// TwinCAT 3 PLC project Motion_Lib
// Title: Motion Library
// Company: Beckhoff UK
// Author: Chris Knight
// ProjectVersion: 4.1.1
// ProgramVersion: 3.1.4026.25
// libraries:
//   Base Library, * (Beckhoff UK)
//   Tc2_MC2, * (Beckhoff Automation GmbH)
//   Tc2_MC2_Drive, * (Beckhoff Automation GmbH)
//   Tc2_Standard, * (Beckhoff Automation GmbH)
//   Tc2_System, * (Beckhoff Automation GmbH)
//   Tc3_Module, * (Beckhoff Automation GmbH)
// project tree:
//   Axis Class/ Axis_Base.TcPOU
//   Interfaces/ I_Axis.TcIO, I_AxisBase.TcIO, I_Status.TcIO, I_Jog.TcIO, I_Position.TcIO, I_Velocity.TcIO
//   Internal/ I_MoveAbs.TcIO, I_MoveMod.TcIO (not stored), I_MoveRel.TcIO, I_MoveVelo.TcIO, MoveAbs.TcPOU, MoveMod.TcPOU, MoveRel.TcPOU, MoveVelo.TcPOU
//   Operations/ GearAxes.TcPOU
//   Project Information/ F_GetCompany.TcPOU, F_GetTitle.TcPOU, F_GetVersion.TcPOU
//   Tasks/ MoveModTask.TcPOU, MoveRelTask.TcPOU, JogTask.TcPOU, CoEResetTask.TcPOU, EnableDisableTask.TcPOU, HaltTask.TcPOU, MoveVeloTask.TcPOU, MoveAbsTask.TcPOU, SoEResetTask.TcPOU
//   Version/ Global_Version.TcGVL

// ---- Version/Global_Version.TcGVL
{attribute 'TcGenerated'}
{attribute 'no-analysis'}
{attribute 'linkalways'}
// This function has been automatically generated from the project information.
VAR_GLOBAL CONSTANT
	{attribute 'const_non_replaced'}
	stLibVersion_Motion_Library : ST_LibVersion := (iMajor := 4, iMinor := 1, iBuild := 1, iRevision := 0, nFlags := 0, sVersion := '4.1.1');
END_VAR

// ---- Interfaces/I_Axis.TcIO
INTERFACE I_Axis EXTENDS I_Cyclic

PROPERTY PUBLIC Acceleration : mc_lreal
GET
END_GET
SET
END_SET
END_PROPERTY

PROPERTY AxisRef : reference to Axis_Ref
GET
END_GET
END_PROPERTY

PROPERTY BufferMode : MC_BufferMode
GET
END_GET
SET
END_SET
END_PROPERTY

PROPERTY PUBLIC Deceleration : mc_lreal
GET
END_GET
SET
END_SET
END_PROPERTY

METHOD PUBLIC DisableAxis : HRESULT
VAR_INPUT
END_VAR
END_METHOD

METHOD PUBLIC EnableAxis : HRESULT
VAR_INPUT
	InhibitPositive : BOOL;
	InhibitNegative : BOOL;
END_VAR
END_METHOD

PROPERTY ErrorID : DWORD
GET
END_GET
END_PROPERTY

METHOD PUBLIC HaltAxis : HRESULT
VAR
END_VAR
END_METHOD

PROPERTY PUBLIC Jerk : mc_lreal
GET
END_GET
SET
END_SET
END_PROPERTY

PROPERTY Operating : BOOL
GET
END_GET
END_PROPERTY

METHOD PUBLIC Reset : HRESULT
VAR
END_VAR
END_METHOD

END_INTERFACE

// ---- Interfaces/I_AxisBase.TcIO
INTERFACE I_AxisBase EXTENDS I_Axis, I_Status

END_INTERFACE

// ---- Interfaces/I_Status.TcIO
INTERFACE I_Status EXTENDS __SYSTEM.IQueryInterface

PROPERTY CurrentPosition : LREAL
GET
END_GET
END_PROPERTY

PROPERTY CurrentVelocity : LREAL
GET
END_GET
END_PROPERTY

PROPERTY ErrorID : DWORD
GET
END_GET
END_PROPERTY

PROPERTY HasError : BOOL
GET
END_GET
END_PROPERTY

PROPERTY InTargetPosition : BOOL
GET
END_GET
END_PROPERTY

PROPERTY InVelocity : BOOL
GET
END_GET
END_PROPERTY

PROPERTY IsCoupled : bool
GET
END_GET
END_PROPERTY

PROPERTY IsEnabled : bool
GET
END_GET
END_PROPERTY

PROPERTY IsStationary : bool
GET
END_GET
END_PROPERTY

END_INTERFACE

// ---- Interfaces/I_Jog.TcIO
INTERFACE I_Jog EXTENDS I_Axis

METHOD Inch : HRESULT
VAR_INPUT
	Distance : MC_LREAL;
	Direction : BOOL;
END_VAR
END_METHOD

METHOD JogFast : HRESULT
VAR_INPUT
	Direction : BOOL;
END_VAR
END_METHOD

METHOD JogSlow : HRESULT
VAR_INPUT
	Direction : BOOL;
END_VAR
END_METHOD

END_INTERFACE

// ---- Interfaces/I_Position.TcIO
INTERFACE I_Position EXTENDS __SYSTEM.IQueryInterface

PROPERTY CurrentPosition : LREAL
GET
END_GET
END_PROPERTY

PROPERTY IsStationary : bool
GET
END_GET
END_PROPERTY

METHOD MoveByDistance : HRESULT
VAR_INPUT
	Distance : MC_LREAL;
	Velocity : MC_LREAL;
END_VAR
END_METHOD

METHOD MoveToModuloPosition : HRESULT
VAR_INPUT
	Position : MC_LREAL;
	Velocity : MC_LREAL;
END_VAR
END_METHOD

METHOD MoveToPosition : HRESULT
VAR_INPUT
	Position : MC_LREAL;
	Velocity : MC_LREAL;
END_VAR
END_METHOD

END_INTERFACE

// ---- Interfaces/I_Velocity.TcIO
INTERFACE I_Velocity

PROPERTY InVelocity : BOOL
GET
END_GET
END_PROPERTY

METHOD MoveAtVelocity : HRESULT
VAR_INPUT
	Direction : MC_Direction;
	Velocity : MC_LREAL;
END_VAR
END_METHOD

END_INTERFACE

// ---- Internal/I_MoveAbs.TcIO
INTERFACE I_MoveAbs

PROPERTY Acceleration : MC_LREAL
GET
END_GET
SET
END_SET
END_PROPERTY

PROPERTY BufferMode : MC_Buffermode
GET
END_GET
SET
END_SET
END_PROPERTY

PROPERTY Busy : BOOL
GET
END_GET
END_PROPERTY

PROPERTY Deceleration : MC_LREAL
GET
END_GET
SET
END_SET
END_PROPERTY

PROPERTY Done : BOOL
GET
END_GET
END_PROPERTY

PROPERTY Error : BOOL
GET
END_GET
END_PROPERTY

PROPERTY Execute : BOOL
GET
END_GET
SET
END_SET
END_PROPERTY

PROPERTY Jerk : MC_LREAL
GET
END_GET
SET
END_SET
END_PROPERTY

PROPERTY Position : MC_LREAL
GET
END_GET
SET
END_SET
END_PROPERTY

PROPERTY Velocity : MC_LREAL
GET
END_GET
SET
END_SET
END_PROPERTY

END_INTERFACE

// ---- Internal/I_MoveRel.TcIO
INTERFACE I_MoveRel

PROPERTY Acceleration : MC_LREAL
GET
END_GET
SET
END_SET
END_PROPERTY

PROPERTY BufferMode : MC_Buffermode
GET
END_GET
SET
END_SET
END_PROPERTY

PROPERTY Busy : BOOL
GET
END_GET
END_PROPERTY

PROPERTY Deceleration : MC_LREAL
GET
END_GET
SET
END_SET
END_PROPERTY

PROPERTY Distance : MC_LREAL
GET
END_GET
SET
END_SET
END_PROPERTY

PROPERTY Done : BOOL
GET
END_GET
END_PROPERTY

PROPERTY Error : BOOL
GET
END_GET
END_PROPERTY

PROPERTY Execute : BOOL
GET
END_GET
SET
END_SET
END_PROPERTY

PROPERTY Jerk : MC_LREAL
GET
END_GET
SET
END_SET
END_PROPERTY

PROPERTY Velocity : MC_LREAL
GET
END_GET
SET
END_SET
END_PROPERTY

END_INTERFACE

// ---- Internal/I_MoveVelo.TcIO
INTERFACE I_MoveVelo

PROPERTY Acceleration : MC_LREAL
GET
END_GET
SET
END_SET
END_PROPERTY

PROPERTY BufferMode : MC_Buffermode
GET
END_GET
SET
END_SET
END_PROPERTY

PROPERTY Busy : BOOL
GET
END_GET
END_PROPERTY

PROPERTY Deceleration : MC_LREAL
GET
END_GET
SET
END_SET
END_PROPERTY

PROPERTY Direction : MC_Direction
GET
END_GET
SET
END_SET
END_PROPERTY

PROPERTY Error : BOOL
GET
END_GET
END_PROPERTY

PROPERTY Execute : BOOL
GET
END_GET
SET
END_SET
END_PROPERTY

PROPERTY InVelocity : BOOL
GET
END_GET
END_PROPERTY

PROPERTY Jerk : MC_LREAL
GET
END_GET
SET
END_SET
END_PROPERTY

PROPERTY Velocity : MC_LREAL
GET
END_GET
SET
END_SET
END_PROPERTY

END_INTERFACE

// ---- Axis Class/Axis_Base.TcPOU
FUNCTION_BLOCK Axis_Base IMPLEMENTS I_AxisBase, I_Axis, I_Position, I_Status, I_Velocity, I_Jog, I_Object, I_Cyclic, I_Resettable
VAR
	_axis : REFERENCE TO Tc2_MC2.AXIS_REF;
	EnableBehaviour : EnableDisableTask;
	DefaultResetBehaviour : CoEResetTask;
	DefaultMoveBehaviour : MoveAbsTask;
	DefaultRelBehaviour : MoveRelTask;
	DefaultModBehaviour : MoveModTask;
	DefaultVeloBehaviour : MoveVeloTask;
	DefaultJogBehaviour : JogTask;
	HaltBehaviour	: HaltTask;
	TaskCollection : ObjectRunner<99>;
	axesReadError : Tc2_MC2.MC_ReadAxisError;
	_ErrorId: DWORD;
	_Operating : BOOL;
	DemandVelo : LREAL;
END_VAR

{analysis -2}

PROPERTY PUBLIC Acceleration : mc_lreal
GET
Acceleration := DefaultMoveBehaviour.Acceleration;
END_GET
SET
DefaultMoveBehaviour.Acceleration := Acceleration;
END_SET
END_PROPERTY

PROPERTY AxisRef : reference to Axis_Ref
GET
AxisRef REF= _axis;
END_GET
END_PROPERTY

PROPERTY BufferMode : MC_BufferMode
GET
BufferMode := DefaultMoveBehaviour.BufferMode;
END_GET
SET
DefaultMoveBehaviour.BufferMode:= BufferMode;
DefaultRelBehaviour.BufferMode := BufferMode;
DefaultModBehaviour.BufferMode := BufferMode;
END_SET
END_PROPERTY

PROPERTY CurrentPosition : LREAL
GET
CurrentPosition := _axis.NcToPlc.ActPos;
END_GET
END_PROPERTY

PROPERTY CurrentVelocity : LREAL
GET
CurrentVelocity := _axis.NcToPlc.ActVelo;
END_GET
END_PROPERTY

METHOD Cycle : HRESULT
VAR_INST
	
END_VAR
_axis.ReadStatus();
axesReadError(Axis := _axis, Enable := TRUE, AxisErrorID => _ErrorId);
TaskCollection.Cycle();

_Operating := DefaultMoveBehaviour.Busy OR DefaultRelBehaviour.Busy OR DefaultModBehaviour.Busy OR DefaultVeloBehaviour.Busy;
END_METHOD

PROPERTY PUBLIC Deceleration : mc_lreal
GET
Deceleration := DefaultMoveBehaviour.Deceleration;
END_GET
SET
DefaultMoveBehaviour.Deceleration := Deceleration;
HaltBehaviour.Deceleration := Deceleration;
END_SET
END_PROPERTY

METHOD PUBLIC DisableAxis : HRESULT
VAR_INPUT
END_VAR
DisableAxis := EnableBehaviour.Disable();
END_METHOD

METHOD PUBLIC EnableAxis : HRESULT
VAR_INPUT
	InhibitPositive : BOOL;
	InhibitNegative : BOOL;
END_VAR
EnableBehaviour.InhibitNegative := InhibitNegative;
EnableBehaviour.InhibitPositive := InhibitPositive;
EnableAxis := EnableBehaviour.Enable();
END_METHOD

PROPERTY ErrorID : DWORD
GET
ErrorId := _ErrorId;
END_GET
END_PROPERTY

//FB_Init is always available implicitly and it is used primarily for initialization.
//The return value is not evaluated. For a specific influence, you can also declare the
//methods explicitly and provide additional code there with the standard initialization
//code. You can evaluate the return value.
METHOD FB_Init: BOOL
VAR_INPUT
    bInitRetains: BOOL; // TRUE: the retain variables are initialized (reset warm / reset cold)
    bInCopyCode: BOOL;  // TRUE: the instance will be copied to the copy code afterward (online change) 
	Axis : Reference TO AXIS_REF;  
END_VAR
EnableBehaviour.AxisRef REF= axis;
DefaultResetBehaviour.AxisRef REF= axis;
DefaultMoveBehaviour.AxisRef REF= axis;
DefaultVeloBehaviour.AxisRef REF= axis;
DefaultJogBehaviour.AxisRef REF= axis;
DefaultRelBehaviour.AxisRef REF= axis;
DefaultModBehaviour.AxisRef REF= axis;
HaltBehaviour.AxisRef REF= axis;
_axis REF= Axis;

DefaultJogBehaviour.RegisterWithParent(Parent := TaskCollection);
DefaultModBehaviour.RegisterWithParent(Parent := TaskCollection);
DefaultMoveBehaviour.RegisterWithParent(Parent := TaskCollection);
DefaultRelBehaviour.RegisterWithParent(Parent := TaskCollection);
DefaultJogBehaviour.RegisterWithParent(Parent := TaskCollection);
DefaultVeloBehaviour.RegisterWithParent(Parent := TaskCollection);
HaltBehaviour.RegisterWithParent(Parent := TaskCollection);
DefaultResetBehaviour.RegisterWithParent(Parent := TaskCollection);
EnableBehaviour.RegisterWithParent(Parent := TaskCollection);
END_METHOD

METHOD PUBLIC HaltAxis : HRESULT
VAR
END_VAR
IF NOT HaltBehaviour.Busy THEN
	HaltAxis := HaltBehaviour.Execute();
	DefaultMoveBehaviour.Abort();
	DefaultVeloBehaviour.Abort();
ELSE 
	HaltAxis := -1;
END_IF
END_METHOD

PROPERTY HasError : BOOL
GET
HasError := _axis.Status.Error;
END_GET
END_PROPERTY

METHOD Inch : HRESULT
VAR_INPUT
	Distance : MC_LREAL;
	Direction : BOOL;
END_VAR
IF FAILED( DefaultJogBehaviour.Inch(Distance, Direction)) THEN
	Inch := -1;
END_IF
END_METHOD

PROPERTY InTargetPosition : BOOL
GET
InTargetPosition := _axis.Status.InTargetPosition;
END_GET
END_PROPERTY

PROPERTY InVelocity : BOOL
GET
InVelocity := ABS(_axis.NcToPlc.ActVelo) < DemandVelo + (DemandVelo * 0.02) AND 
				ABS(_axis.NcToPlc.ActVelo) > DemandVelo - (DemandVelo * 0.02);
END_GET
END_PROPERTY

PROPERTY IsCoupled : bool
GET
isCoupled := _axis.Status.Coupled;
END_GET
END_PROPERTY

PROPERTY IsEnabled : bool
GET
isEnabled := not _axis.Status.Disabled;
END_GET
END_PROPERTY

PROPERTY IsStationary : bool
GET
isStationary := NOT _axis.Status.HasJob AND _axis.Status.NotMoving;
END_GET
END_PROPERTY

PROPERTY PUBLIC Jerk : mc_lreal
GET
Jerk := DefaultMoveBehaviour.Jerk;
END_GET
SET
DefaultMoveBehaviour.Jerk := Jerk;
HaltBehaviour.Jerk := Jerk;
END_SET
END_PROPERTY

METHOD JogFast : HRESULT
VAR_INPUT
	Direction : BOOL;
END_VAR
IF FAILED(DefaultJogBehaviour.JogFast(Direction)) THEN
	JogFast := -1;
END_IF
END_METHOD

METHOD JogSlow : HRESULT
VAR_INPUT
	Direction : BOOL;
END_VAR
IF FAILED(DefaultJogBehaviour.JogSlow(Direction)) THEN
	JogSlow := -1;
END_IF
END_METHOD

METHOD MoveAtVelocity : HRESULT
VAR_INPUT
	Direction : MC_Direction;
	Velocity : MC_LREAL;
END_VAR
IF Velocity = 0 THEN 
	MoveAtVelocity := -1;
	RETURN;
END_IF

IF SUCCEEDED(DefaultVeloBehaviour.MoveAtVelocity(Direction, Velocity)) THEN
	DemandVelo := Velocity;
ELSE
	MoveAtVelocity := -1;
END_IF
END_METHOD

METHOD MoveByDistance : HRESULT
VAR_INPUT
	Distance : MC_LREAL;
	Velocity : MC_LREAL;
END_VAR
IF ABS(Distance) = 0 THEN
	MoveByDistance := -1;
	RETURN;
END_IF
IF _axis.Status.Disabled THEN
	MoveByDistance := -2;
	RETURN;
END_IF

IF _axis.Status.Error THEN
	MoveByDistance := -3;
	RETURN;
END_IF

DefaultRelBehaviour.MoveBy(Distance,Velocity);
END_METHOD

METHOD MoveToModuloPosition : HRESULT
VAR_INPUT
	Position : MC_LREAL;
	Velocity : MC_LREAL;
END_VAR
IF Velocity = 0 THEN
	MoveToModuloPosition := -1;
	RETURN;
END_IF

IF _axis.Status.Disabled THEN
	MoveToModuloPosition := -2;
	RETURN;
END_IF

IF _axis.Status.Error THEN
	MoveToModuloPosition := -3;
	RETURN;
END_IF

DefaultModBehaviour.MoveTo(Position,Velocity);
END_METHOD

METHOD PUBLIC MoveToPosition : HRESULT
VAR_INPUT
	Position : MC_LREAL;
	Velocity : MC_LREAL;
END_VAR
IF Velocity = 0 THEN
	Base_Library.Tracing.Trace.Warning(TO_STRING(_axis.NcToPlc.AxisId), 'Abs Move Fail - 0 Velo');
	MoveToPosition := -1;
	RETURN;
END_IF

IF _axis.Status.Disabled THEN
	Base_Library.Tracing.Trace.Warning(TO_STRING(_axis.NcToPlc.AxisId), 'Abs Move Fail - Disabled');
	MoveToPosition := -2;
	RETURN;
END_IF

IF _axis.Status.Error THEN
	Base_Library.Tracing.Trace.Warning(TO_STRING(_axis.NcToPlc.AxisId), 'Abs Move Fail - Error');
	MoveToPosition := -3;
	RETURN;
END_IF

Base_Library.Tracing.Trace.Verbose(TO_STRING(_axis.NcToPlc.AxisId), 'Abs Move Success');
DefaultMoveBehaviour.MoveTo(Position,Velocity);
END_METHOD

PROPERTY Operating : BOOL
GET
Operating := _Operating;
END_GET
END_PROPERTY

METHOD RegisterWithParent
VAR_INPUT
	Parent	: Base_Library.I_HostObjects;
END_VAR
Parent.RegisterCyclic(THIS^);
Parent.RegisterResettable(THIS^);
END_METHOD

METHOD PUBLIC Reset : HRESULT
VAR
	ResetResult : HRESULT;
	MoveAbortResult : BOOL;
	HaltAbortResult : BOOL;
END_VAR
TaskCollection.Reset();
//TaskCollection.Abort();
END_METHOD

END_FUNCTION_BLOCK

// ---- Tasks/EnableDisableTask.TcPOU
FUNCTION_BLOCK EnableDisableTask IMPLEMENTS I_Task, I_Cyclic, I_Object, I_Abortable
VAR
	mcPower : Tc2_MC2.MC_Power;
	_Axis : REFERENCE TO Tc2_MC2.AXIS_REF;
	_InhibitPos : BOOL := FALSE;
	_InhibitNeg : BOOL := FALSE;
END_VAR

{analysis -2}

METHOD Abort : HRESULT
mcPower.Enable := FALSE;
mcPower.Enable_Negative := FALSE;
mcPower.Enable_Positive := FALSE;
END_METHOD

PROPERTY AxisRef : reference to Axis_Ref
GET // PUBLIC
AxisRef REF= _Axis;
END_GET
SET
_Axis REF= AxisRef;
END_SET
END_PROPERTY

PROPERTY Busy : BOOL
GET
Busy := mcPower.Busy;
END_GET
END_PROPERTY

METHOD Cycle : HRESULT
VAR_INPUT
END_VAR
mcPower(Axis := _Axis);
END_METHOD

METHOD Disable : HRESULT
VAR_INPUT
END_VAR
IF NOT mcPower.Enable THEN
	Disable := -1;
ELSE
	mcPower.Enable := FALSE;
END_IF
END_METHOD

PROPERTY Done : BOOL
GET
Done := NOT mcPower.Busy;
END_GET
END_PROPERTY

METHOD Enable : HRESULT
VAR_INPUT
END_VAR
IF mcPower.Enable THEN 
	Enable := -1;
ELSE
	mcPower.Enable := TRUE;
	mcPower.Enable_Negative := NOT _InhibitNeg;
	mcPower.Enable_Positive := NOT _InhibitPos;
END_IF
END_METHOD

PROPERTY Error : BOOL
GET
Error := mcPower.Error;
END_GET
END_PROPERTY

PROPERTY InhibitNegative : BOOL
GET
InhibitNegative := _InhibitNeg;
END_GET
SET
_InhibitNeg := InhibitNegative;
END_SET
END_PROPERTY

PROPERTY InhibitPositive : BOOL
GET
InhibitPositive := _InhibitPos;
END_GET
SET
_InhibitPos := InhibitPositive;
END_SET
END_PROPERTY

METHOD RegisterWithParent
VAR_INPUT
	Parent	: I_HostObjects;
END_VAR
Parent.RegisterAbortable(THIS^);
Parent.RegisterCyclic(THIS^);
Parent.RegisterTask(THIS^);
END_METHOD

END_FUNCTION_BLOCK

// ---- Tasks/CoEResetTask.TcPOU
FUNCTION_BLOCK CoEResetTask IMPLEMENTS I_Task, I_Cyclic, I_Object, I_Abortable, I_Abortable, I_Resettable
VAR
	mcReset : Tc2_MC2.MC_Reset;
	_Axis : REFERENCE TO Tc2_MC2.AXIS_REF;
END_VAR

{analysis -2}

METHOD Abort : HRESULT
mcReset.Execute := FALSE;
END_METHOD

PROPERTY AxisRef : reference to Axis_Ref
GET // PUBLIC
AxisRef REF= _Axis;
END_GET
SET
_Axis REF= AxisRef;
END_SET
END_PROPERTY

PROPERTY Busy : BOOL
GET
Busy := mcReset.Busy;
END_GET
END_PROPERTY

METHOD Cycle : HRESULT
VAR_INPUT
END_VAR
mcReset(Axis := _Axis);
mcReset.Execute := FALSE;
END_METHOD

PROPERTY Done : BOOL
GET
Done := mcReset.Done;
END_GET
END_PROPERTY

PROPERTY Error : BOOL
GET
Error := mcReset.Error;
END_GET
END_PROPERTY

METHOD RegisterWithParent
VAR_INPUT
	Parent	: I_HostObjects;
END_VAR
Parent.RegisterAbortable(THIS^);
Parent.RegisterCyclic(THIS^);
Parent.RegisterTask(THIS^);
Parent.RegisterResettable(THIS^);
END_METHOD

METHOD Reset : HRESULT
VAR_INPUT
END_VAR
IF mcReset.Execute THEN
	Reset := -1;
ELSE
	mcReset.Execute := TRUE;
END_IF
END_METHOD

END_FUNCTION_BLOCK

// ---- Tasks/MoveAbsTask.TcPOU
FUNCTION_BLOCK MoveAbsTask IMPLEMENTS I_Task, I_Cyclic, I_Object, I_Abortable
VAR_INPUT
END_VAR
VAR_OUTPUT
END_VAR
VAR
	moveAbs : ARRAY[0..1] OF MoveAbs;
	iMoveAbs : I_MoveAbs := MoveAbs[0];
	moveIndex : INT;
	_Axis : REFERENCE TO AXIS_REF;
END_VAR

{analysis -2}

METHOD Abort : HRESULT
iMoveAbs.Execute := FALSE;
iMoveAbs.Position := 0;
iMoveAbs.Velocity := 0;
END_METHOD

PROPERTY PUBLIC Acceleration : mc_lreal
GET
Acceleration := moveAbs[0].Acceleration;
END_GET
SET
MoveAbs[0].Acceleration := Acceleration;
MoveAbs[1].Acceleration := Acceleration;
END_SET
END_PROPERTY

PROPERTY AxisRef : reference to Axis_Ref
GET // PUBLIC
AxisRef REF= _Axis;
END_GET
SET
_Axis REF= AxisRef;
END_SET
END_PROPERTY

PROPERTY BufferMode : MC_BufferMode
GET
BufferMode := MoveAbs[0].BufferMode;
END_GET
SET
MoveAbs[0].BufferMode := BufferMode;
MoveAbs[1].BufferMode := BufferMode;
END_SET
END_PROPERTY

PROPERTY Busy : BOOL
GET
Busy := iMoveAbs.Busy;
END_GET
END_PROPERTY

METHOD Cycle : HRESULT
VAR_INPUT
END_VAR
moveAbs[0](Axis := _Axis);
moveAbs[1](Axis := _Axis);

iMoveAbs.Execute := FALSE;
END_METHOD

PROPERTY PUBLIC Deceleration : mc_lreal
GET
Deceleration := MoveAbs[0].Deceleration;
END_GET
SET
MoveAbs[0].Deceleration := Deceleration;
MoveAbs[1].Deceleration := Deceleration;
END_SET
END_PROPERTY

PROPERTY Done : BOOL
GET
Done := iMoveAbs.Done;
END_GET
END_PROPERTY

PROPERTY Error : BOOL
GET
Error := iMoveAbs.Error;
END_GET
END_PROPERTY

PROPERTY PUBLIC Jerk : mc_lreal
GET
Jerk := MoveAbs[0].Jerk;
END_GET
SET
MoveAbs[0].Jerk := Jerk;
MoveAbs[1].Jerk := Jerk;
END_SET
END_PROPERTY

METHOD MoveTo : HRESULT
VAR_INPUT
	Position : MC_LREAL;
	Velocity : MC_LREAL;
END_VAR
IF Velocity <= 0.0 THEN
	MoveTo := -1;
	RETURN;
END_IF
Abort();
IF moveIndex = 0 THEN
	moveIndex := 1;
ELSE
	moveIndex := 0;
END_IF
iMoveAbs := moveAbs[moveIndex];
iMoveAbs.Execute := TRUE;
iMoveAbs.Position := Position;
iMoveAbs.Velocity := Velocity;
END_METHOD

METHOD RegisterWithParent
VAR_INPUT
	Parent	: I_HostObjects;
END_VAR
Parent.RegisterAbortable(THIS^);
Parent.RegisterCyclic(THIS^);
Parent.RegisterTask(THIS^);
END_METHOD

END_FUNCTION_BLOCK

// ---- Internal/MoveAbs.TcPOU
FUNCTION_BLOCK MoveAbs IMPLEMENTS I_MoveAbs
VAR
	mcMoveAbs : MC_MoveAbsolute;
END_VAR
VAR_IN_OUT
	Axis : AXIS_REF;
END_VAR

mcMoveAbs(Axis := Axis);

PROPERTY Acceleration : MC_LREAL
GET
Acceleration := mcMoveAbs.Acceleration;
END_GET
SET
mcMoveAbs.Acceleration := Acceleration;
END_SET
END_PROPERTY

PROPERTY BufferMode : MC_Buffermode
GET
BufferMode := mcMoveAbs.BufferMode;
END_GET
SET
mcMoveAbs.BufferMode := BufferMode;
END_SET
END_PROPERTY

PROPERTY Busy : BOOL
GET
Busy := mcMoveAbs.Busy;
END_GET
END_PROPERTY

PROPERTY Deceleration : MC_LREAL
GET
Deceleration := mcMoveAbs.Deceleration;
END_GET
SET
mcMoveAbs.Deceleration := Deceleration;
END_SET
END_PROPERTY

PROPERTY Done : BOOL
GET
Done := mcMoveAbs.Done;
END_GET
END_PROPERTY

PROPERTY Error : BOOL
GET
Error := mcMoveAbs.Error;
END_GET
END_PROPERTY

PROPERTY Execute : BOOL
GET
Execute := mcMoveAbs.Execute;
END_GET
SET
mcMoveAbs.Execute := Execute;
END_SET
END_PROPERTY

PROPERTY Jerk : MC_LREAL
GET
Jerk := mcMoveAbs.Jerk;
END_GET
SET
mcMoveAbs.Jerk := Jerk;
END_SET
END_PROPERTY

PROPERTY Position : MC_LREAL
GET
Position := mcMoveAbs.Position;
END_GET
SET
mcMoveAbs.Position := Position;
END_SET
END_PROPERTY

PROPERTY Velocity : MC_LREAL
GET
Velocity := mcMoveAbs.Velocity;
END_GET
SET
mcMoveAbs.Velocity := Velocity;
END_SET
END_PROPERTY

END_FUNCTION_BLOCK

// ---- Tasks/MoveRelTask.TcPOU
FUNCTION_BLOCK MoveRelTask IMPLEMENTS I_Task, I_Cyclic, I_Object, I_Abortable
VAR_INPUT
END_VAR
VAR_OUTPUT
END_VAR
VAR
	moveRel : ARRAY[0..1] OF MoveRel;
	iMoveRel : I_MoveRel := moveRel[0];
	moveIndex : INT;
	_Axis : REFERENCE TO AXIS_REF;
END_VAR

{analysis -2}

METHOD Abort : HRESULT
iMoveRel.Execute := FALSE;
iMoveRel.Distance := 0;
iMoveRel.Velocity := 0;
END_METHOD

PROPERTY PUBLIC Acceleration : mc_lreal
GET
Acceleration := moveRel[0].Acceleration;
END_GET
SET
moveRel[0].Acceleration := Acceleration;
moveRel[1].Acceleration := Acceleration;
END_SET
END_PROPERTY

PROPERTY AxisRef : reference to Axis_Ref
GET // PUBLIC
AxisRef REF= _Axis;
END_GET
SET
_Axis REF= AxisRef;
END_SET
END_PROPERTY

PROPERTY BufferMode : MC_BufferMode
GET
BufferMode := moveRel[0].BufferMode;
END_GET
SET
moveRel[0].BufferMode := BufferMode;
moveRel[1].BufferMode := BufferMode;
END_SET
END_PROPERTY

PROPERTY Busy : BOOL
GET
Busy := iMoveRel.Busy;
END_GET
END_PROPERTY

METHOD Cycle : HRESULT
VAR_INPUT
END_VAR
moveRel[0](Axis := _Axis);
moveRel[1](Axis := _Axis);

iMoveRel.Execute := FALSE;
END_METHOD

PROPERTY PUBLIC Deceleration : mc_lreal
GET
Deceleration := moveRel[0].Deceleration;
END_GET
SET
moveRel[0].Deceleration := Deceleration;
moveRel[1].Deceleration := Deceleration;
END_SET
END_PROPERTY

PROPERTY Done : BOOL
GET
Done := iMoveRel.Done;
END_GET
END_PROPERTY

PROPERTY Error : BOOL
GET
Error := iMoveRel.Error;
END_GET
END_PROPERTY

PROPERTY PUBLIC Jerk : mc_lreal
GET
Jerk := moveRel[0].Jerk;
END_GET
SET
moveRel[0].Jerk := Jerk;
moveRel[1].Jerk := Jerk;
END_SET
END_PROPERTY

METHOD MoveBy : HRESULT
VAR_INPUT
	Distance : MC_LREAL;
	Velocity : MC_LREAL;
END_VAR
IF Velocity <= 0.0 THEN
	MoveBy := -1;
	RETURN;
END_IF
Abort();
IF moveIndex = 0 THEN
	moveIndex := 1;
ELSE
	moveIndex := 0;
END_IF
iMoveRel := moveRel[moveIndex];
iMoveRel.Distance := Distance;
iMoveRel.Velocity := Velocity;
iMoveRel.Execute := TRUE;
END_METHOD

METHOD RegisterWithParent
VAR_INPUT
	Parent	: I_HostObjects;
END_VAR
Parent.RegisterAbortable(THIS^);
Parent.RegisterCyclic(THIS^);
Parent.RegisterTask(THIS^);
END_METHOD

END_FUNCTION_BLOCK

// ---- Internal/MoveRel.TcPOU
FUNCTION_BLOCK MoveRel IMPLEMENTS I_MoveRel
VAR
	mcMoveRel : MC_MoveRelative;
END_VAR
VAR_IN_OUT
	Axis : AXIS_REF;
END_VAR

mcMoveRel(Axis := Axis);

PROPERTY Acceleration : MC_LREAL
GET
Acceleration := mcMoveRel.Acceleration;
END_GET
SET
mcMoveRel.Acceleration := Acceleration;
END_SET
END_PROPERTY

PROPERTY BufferMode : MC_Buffermode
GET
BufferMode := mcMoveRel.BufferMode;
END_GET
SET
mcMoveRel.BufferMode := BufferMode;
END_SET
END_PROPERTY

PROPERTY Busy : BOOL
GET
Busy := mcMoveRel.Busy;
END_GET
END_PROPERTY

PROPERTY Deceleration : MC_LREAL
GET
Deceleration := mcMoveRel.Deceleration;
END_GET
SET
mcMoveRel.Deceleration := Deceleration;
END_SET
END_PROPERTY

PROPERTY Distance : MC_LREAL
GET
Distance := mcMoveRel.Distance;
END_GET
SET
mcMoveRel.Distance := Distance;
END_SET
END_PROPERTY

PROPERTY Done : BOOL
GET
Done := mcMoveRel.Done;
END_GET
END_PROPERTY

PROPERTY Error : BOOL
GET
Error := mcMoveRel.Error;
END_GET
END_PROPERTY

PROPERTY Execute : BOOL
GET
Execute := mcMoveRel.Execute;
END_GET
SET
mcMoveRel.Execute := Execute;
END_SET
END_PROPERTY

PROPERTY Jerk : MC_LREAL
GET
Jerk := mcMoveRel.Jerk;
END_GET
SET
mcMoveRel.Jerk := Jerk;
END_SET
END_PROPERTY

PROPERTY Velocity : MC_LREAL
GET
Velocity := mcMoveRel.Velocity;
END_GET
SET
mcMoveRel.Velocity := Velocity;
END_SET
END_PROPERTY

END_FUNCTION_BLOCK

// ---- Tasks/MoveModTask.TcPOU
FUNCTION_BLOCK MoveModTask IMPLEMENTS I_Task, I_Cyclic, I_Object, I_Abortable
VAR_INPUT
END_VAR
VAR_OUTPUT
END_VAR
VAR
	moveMod : ARRAY[0..1] OF MoveMod;
	iMoveMod : I_MoveMod := moveMod[0];
	moveIndex : INT;
	_Axis : REFERENCE TO AXIS_REF;
END_VAR

{analysis -2}

METHOD Abort : HRESULT
iMoveMod.Execute := FALSE;
iMoveMod.Position := 0;
iMoveMod.Velocity := 0;
END_METHOD

PROPERTY PUBLIC Acceleration : mc_lreal
GET
Acceleration := moveMod[0].Acceleration;
END_GET
SET
moveMod[0].Acceleration := Acceleration;
moveMod[1].Acceleration := Acceleration;
END_SET
END_PROPERTY

PROPERTY AxisRef : reference to Axis_Ref
GET // PUBLIC
AxisRef REF= _Axis;
END_GET
SET
_Axis REF= AxisRef;
END_SET
END_PROPERTY

PROPERTY BufferMode : MC_BufferMode
GET
BufferMode := moveMod[0].BufferMode;
END_GET
SET
moveMod[0].BufferMode := BufferMode;
moveMod[1].BufferMode := BufferMode;
END_SET
END_PROPERTY

PROPERTY Busy : BOOL
GET
Busy := iMoveMod.Busy;
END_GET
END_PROPERTY

METHOD Cycle : HRESULT
VAR_INPUT
END_VAR
moveMod[0](Axis := _Axis);
moveMod[1](Axis := _Axis);

iMoveMod.Execute := FALSE;
END_METHOD

PROPERTY PUBLIC Deceleration : mc_lreal
GET
Deceleration := moveMod[0].Deceleration;
END_GET
SET
moveMod[0].Deceleration := Deceleration;
moveMod[1].Deceleration := Deceleration;
END_SET
END_PROPERTY

PROPERTY Done : BOOL
GET
Done := iMoveMod.Done;
END_GET
END_PROPERTY

PROPERTY Error : BOOL
GET
Error := iMoveMod.Error;
END_GET
END_PROPERTY

PROPERTY PUBLIC Jerk : mc_lreal
GET
Jerk := moveMod[0].Jerk;
END_GET
SET
moveMod[0].Jerk := Jerk;
moveMod[1].Jerk := Jerk;
END_SET
END_PROPERTY

METHOD MoveTo : hresult
VAR_INPUT
	Position : MC_LREAL;
	Velocity : MC_LREAL;
END_VAR
IF Velocity <= 0.0 THEN
	MoveTo := -1;
	RETURN;
END_IF
Abort();
IF moveIndex = 0 THEN
	moveIndex := 1;
ELSE
	moveIndex := 0;
END_IF
iMoveMod := moveMod[moveIndex];

iMoveMod.Position := Position;
iMoveMod.Velocity := Velocity;
iMoveMod.Execute := TRUE;
END_METHOD

METHOD RegisterWithParent
VAR_INPUT
	Parent	: I_HostObjects;
END_VAR
Parent.RegisterAbortable(THIS^);
Parent.RegisterCyclic(THIS^);
Parent.RegisterTask(THIS^);
END_METHOD

END_FUNCTION_BLOCK

// ---- Internal/MoveMod.TcPOU
FUNCTION_BLOCK MoveMod IMPLEMENTS I_MoveMod
VAR
	mcMoveMod : MC_MoveModulo;
END_VAR
VAR_IN_OUT
	Axis : AXIS_REF;
END_VAR

mcMoveMod(Axis := Axis);

PROPERTY Acceleration : MC_LREAL
GET
Acceleration := mcMoveMod.Acceleration;
END_GET
SET
mcMoveMod.Acceleration := Acceleration;
END_SET
END_PROPERTY

PROPERTY BufferMode : MC_Buffermode
GET
BufferMode := mcMoveMod.BufferMode;
END_GET
SET
mcMoveMod.BufferMode := BufferMode;
END_SET
END_PROPERTY

PROPERTY Busy : BOOL
GET
Busy := mcMoveMod.Busy;
END_GET
END_PROPERTY

PROPERTY Deceleration : MC_LREAL
GET
Deceleration := mcMoveMod.Deceleration;
END_GET
SET
mcMoveMod.Deceleration := Deceleration;
END_SET
END_PROPERTY

PROPERTY Done : BOOL
GET
Done := mcMoveMod.Done;
END_GET
END_PROPERTY

PROPERTY Error : BOOL
GET
Error := mcMoveMod.Error;
END_GET
END_PROPERTY

PROPERTY Execute : BOOL
GET
Execute := mcMoveMod.Execute;
END_GET
SET
mcMoveMod.Execute := Execute;
END_SET
END_PROPERTY

PROPERTY Jerk : MC_LREAL
GET
Jerk := mcMoveMod.Jerk;
END_GET
SET
mcMoveMod.Jerk := Jerk;
END_SET
END_PROPERTY

PROPERTY Position : MC_LREAL
GET
Position := mcMoveMod.Position;
END_GET
SET
mcMoveMod.Position := Position;
END_SET
END_PROPERTY

PROPERTY Velocity : MC_LREAL
GET
Velocity := mcMoveMod.Velocity;
END_GET
SET
mcMoveMod.Velocity := Velocity;
END_SET
END_PROPERTY

END_FUNCTION_BLOCK

// ---- Tasks/MoveVeloTask.TcPOU
FUNCTION_BLOCK MoveVeloTask IMPLEMENTS I_Task, I_Cyclic, I_Object, I_Abortable
VAR
	mcMoveVelo : ARRAY[0..1] OF MoveVelo;
	iMoveVelo : I_MoveVelo := mcMoveVelo[0];
	moveIndex : INT;
	_Axis : REFERENCE TO AXIS_REF;
END_VAR

METHOD Abort : HRESULT
iMoveVelo.Execute := FALSE;
iMoveVelo.Velocity := 0;
END_METHOD

PROPERTY PUBLIC Acceleration : mc_lreal
GET
Acceleration := mcMoveVelo[0].Acceleration;
END_GET
SET
IF Acceleration >= 0.0 THEN
	mcMoveVelo[0].Acceleration := Acceleration;
	mcMoveVelo[1].Acceleration := Acceleration;
END_IF
END_SET
END_PROPERTY

PROPERTY AxisRef : reference to Axis_Ref
GET // PUBLIC
AxisRef REF= _Axis;
END_GET
SET
_Axis REF= AxisRef;
END_SET
END_PROPERTY

PROPERTY BufferMode : MC_BufferMode
GET
BufferMode := mcMoveVelo[0].BufferMode;
END_GET
SET
mcMoveVelo[0].BufferMode := BufferMode;
mcMoveVelo[1].BufferMode := BufferMode;
END_SET
END_PROPERTY

PROPERTY Busy : BOOL
GET
Busy := iMoveVelo.Busy;
END_GET
END_PROPERTY

METHOD Cycle : HRESULT
mcMoveVelo[0](Axis := _Axis);
mcMoveVelo[1](Axis := _Axis);

iMoveVelo.Execute := FALSE;
END_METHOD

PROPERTY Deceleration : MC_LREAL
GET
Deceleration := mcMoveVelo[0].Deceleration;
END_GET
SET
IF Deceleration >= 0.0 THEN
	mcMoveVelo[0].Deceleration := Deceleration;
	mcMoveVelo[1].Deceleration := Deceleration;
END_IF
END_SET
END_PROPERTY

PROPERTY Done : BOOL
GET
Done := NOT iMoveVelo.Busy;
END_GET
END_PROPERTY

PROPERTY Error : BOOL
GET
Error := iMoveVelo.Error;
END_GET
END_PROPERTY

PROPERTY Jerk : MC_LREAL
GET
Jerk := mcMoveVelo[0].Jerk;
END_GET
SET
IF Jerk >= 0.0 THEN
	mcMoveVelo[0].Jerk := Jerk;
	mcMoveVelo[1].Jerk := Jerk;
END_IF
END_SET
END_PROPERTY

METHOD MoveAtVelocity : HRESULT
VAR_INPUT
	Direction : MC_Direction;
	Velocity : MC_LREAL;
END_VAR
IF Velocity <= 0 THEN
	MoveAtVelocity := -1;
	RETURN;
END_IF

Abort();
IF moveIndex = 0 THEN
	moveIndex := 1;
ELSE
	moveIndex := 0;
END_IF
iMoveVelo := mcMoveVelo[moveIndex];
iMoveVelo.Direction := Direction;
iMoveVelo.Velocity := Velocity;
iMoveVelo.Execute := TRUE;
END_METHOD

METHOD RegisterWithParent
VAR_INPUT
	Parent	: I_HostObjects;
END_VAR
Parent.RegisterAbortable(THIS^);
Parent.RegisterCyclic(THIS^);
Parent.RegisterTask(THIS^);
END_METHOD

END_FUNCTION_BLOCK

// ---- Internal/MoveVelo.TcPOU
FUNCTION_BLOCK MoveVelo IMPLEMENTS I_MoveVelo
VAR
	mcMoveVelo : MC_MoveVelocity;
END_VAR
VAR_IN_OUT
	Axis : AXIS_REF;
END_VAR

mcMoveVelo(Axis := Axis);

PROPERTY Acceleration : MC_LREAL
GET
Acceleration := mcMoveVelo.Acceleration;
END_GET
SET
mcMoveVelo.Acceleration := Acceleration;
END_SET
END_PROPERTY

PROPERTY BufferMode : MC_Buffermode
GET
BufferMode := mcMoveVelo.BufferMode;
END_GET
SET
mcMoveVelo.BufferMode := BufferMode;
END_SET
END_PROPERTY

PROPERTY Busy : BOOL
GET
Busy := mcMoveVelo.Busy;
END_GET
END_PROPERTY

PROPERTY Deceleration : MC_LREAL
GET
Deceleration := mcMoveVelo.Deceleration;
END_GET
SET
mcMoveVelo.Deceleration := Deceleration;
END_SET
END_PROPERTY

PROPERTY Direction : MC_Direction
GET
Direction := mcMoveVelo.Direction;
END_GET
SET
mcMoveVelo.Direction := Direction;
END_SET
END_PROPERTY

PROPERTY Error : BOOL
GET
Error := mcMoveVelo.Error;
END_GET
END_PROPERTY

PROPERTY Execute : BOOL
GET
Execute := mcMoveVelo.Execute;
END_GET
SET
mcMoveVelo.Execute := Execute;
END_SET
END_PROPERTY

PROPERTY InVelocity : BOOL
GET
InVelocity := mcMoveVelo.InVelocity;
END_GET
END_PROPERTY

PROPERTY Jerk : MC_LREAL
GET
Jerk := mcMoveVelo.Jerk;
END_GET
SET
mcMoveVelo.Jerk := Jerk;
END_SET
END_PROPERTY

PROPERTY Velocity : MC_LREAL
GET
Velocity := mcMoveVelo.Velocity;
END_GET
SET
mcMoveVelo.Velocity := Velocity;
END_SET
END_PROPERTY

END_FUNCTION_BLOCK

// ---- Tasks/JogTask.TcPOU
FUNCTION_BLOCK JogTask IMPLEMENTS I_Task, I_Cyclic, I_Object, I_Abortable
VAR
	mcJog : MC_Jog;
	_Axis : REFERENCE TO Tc2_MC2.AXIS_REF;
END_VAR

METHOD Abort : HRESULT
mcJog.JogBackwards := FALSE;
mcJog.JogForward := FALSE;
END_METHOD

PROPERTY PUBLIC Acceleration : mc_lreal
GET
Acceleration := mcJog.Acceleration;
END_GET
SET
IF Acceleration >= 0.0 THEN
	mcJog.Acceleration := Acceleration;
END_IF
END_SET
END_PROPERTY

PROPERTY AxisRef : reference to Axis_Ref
GET // PUBLIC
AxisRef REF= _Axis;
END_GET
SET
_Axis REF= AxisRef;
END_SET
END_PROPERTY

PROPERTY Busy : BOOL
GET
Busy := mcJog.Busy;
END_GET
END_PROPERTY

METHOD Cycle : HRESULT
mcJog(Axis := _Axis);
IF mcJog.JogBackwards OR mcJog.JogForward THEN
	mcJog.JogForward := FALSE;
	mcJog.JogBackwards := FALSE;
END_IF
END_METHOD

PROPERTY Deceleration : MC_LREAL
GET
Deceleration := mcJog.Deceleration;
END_GET
SET
IF Deceleration >= 0.0 THEN
	mcJog.Deceleration := Deceleration;
END_IF
END_SET
END_PROPERTY

PROPERTY Done : BOOL
GET
Done := mcJog.Done;
END_GET
END_PROPERTY

PROPERTY Error : BOOL
GET
Error := mcJog.Error;
END_GET
END_PROPERTY

METHOD Inch : HRESULT
VAR_INPUT
	Distance : MC_LREAL;
	Direction : BOOL;
END_VAR
IF Distance > 0.0 AND NOT mcJog.Busy THEN
	mcJog.Mode := E_JogMode.MC_JOGMODE_INCHING;
	IF Direction THEN
		mcJog.JogForward := TRUE;
	ELSE
		mcJog.JogBackwards := TRUE;
	END_IF
	Inch := 1;
ELSE
	Inch := -1;
END_IF
END_METHOD

PROPERTY Jerk : MC_LREAL
GET
Jerk := mcJog.Jerk;
END_GET
SET
IF Jerk >= 0.0 THEN
	mcJog.Jerk := Jerk;
END_IF
END_SET
END_PROPERTY

METHOD JogFast : HRESULT
VAR_INPUT
	Direction : BOOL;
END_VAR
mcJog.Mode := E_JogMode.MC_JOGMODE_STANDARD_FAST;
IF Direction THEN
	mcJog.JogForward := TRUE;
ELSE
	mcJog.JogBackwards := TRUE;
END_IF
JogFast := 1;
END_METHOD

METHOD JogSlow : HRESULT
VAR_INPUT
	Direction : BOOL;
END_VAR
mcJog.Mode := E_JogMode.MC_JOGMODE_STANDARD_SLOW;
IF Direction THEN
	mcJog.JogForward := TRUE;
ELSE
	mcJog.JogBackwards := TRUE;
END_IF
JogSlow := 1;
END_METHOD

METHOD RegisterWithParent
VAR_INPUT
	Parent	: I_HostObjects;
END_VAR
Parent.RegisterAbortable(THIS^);
Parent.RegisterCyclic(THIS^);
Parent.RegisterTask(THIS^);
END_METHOD

END_FUNCTION_BLOCK

// ---- Tasks/HaltTask.TcPOU
FUNCTION_BLOCK HaltTask IMPLEMENTS I_Task, I_Cyclic, I_Abortable, I_Object
VAR_INPUT
END_VAR
VAR_OUTPUT
END_VAR
VAR
	mcHalt : Tc2_MC2.MC_Halt;
	_Axis : REFERENCE TO Tc2_MC2.AXIS_REF;
END_VAR

{analysis -2}

METHOD Abort : HRESULT
mcHalt.Execute := FALSE;
END_METHOD

PROPERTY AxisRef : reference to Axis_Ref
GET // PUBLIC
AxisRef REF= _Axis;
END_GET
SET
_Axis REF= AxisRef;
END_SET
END_PROPERTY

PROPERTY Busy : BOOL
GET
Busy := mcHalt.Busy;
END_GET
END_PROPERTY

METHOD Cycle : HRESULT
VAR_INPUT
END_VAR
mcHalt(Axis := _Axis);
mcHalt.Execute := FALSE;
END_METHOD

PROPERTY Deceleration : MC_LREAL
GET
Deceleration := mcHalt.Deceleration;
END_GET
SET
IF Deceleration >= 0.0 THEN
	mcHalt.Deceleration := Deceleration;
END_IF
END_SET
END_PROPERTY

PROPERTY Done : BOOL
GET
Done := mcHalt.Done;
END_GET
END_PROPERTY

PROPERTY Error : BOOL
GET
Error := mcHalt.Error;
END_GET
END_PROPERTY

METHOD Execute : HRESULT
VAR_INPUT
END_VAR
IF _Axis.Status.Moving AND NOT mcHalt.Execute THEN
	Execute := S_OK;
	mcHalt.Execute := TRUE;
ELSE
	Execute := S_FALSE;
END_IF
END_METHOD

PROPERTY Jerk : MC_LREAL
GET
Jerk := mcHalt.Jerk;
END_GET
SET
IF Jerk >= 0.0 THEN
	mcHalt.Jerk := Jerk;
END_IF
END_SET
END_PROPERTY

METHOD RegisterWithParent
VAR_INPUT
	Parent	: I_HostObjects;
END_VAR
Parent.RegisterAbortable(THIS^);
Parent.RegisterCyclic(THIS^);
Parent.RegisterTask(THIS^);
END_METHOD

END_FUNCTION_BLOCK

// ---- Operations/GearAxes.TcPOU
FUNCTION_BLOCK GearAxes IMPLEMENTS I_Object, I_Abortable, I_Cyclic
VAR
	mcGearIn : MC_GearIn;
	mcGearOut : MC_GearOut;
	_AxisMaster : I_AxisBase;
	_AxisSlave : I_AxisBase;
END_VAR

METHOD Abort : HRESULT
mcGearIn.Execute := FALSE;
mcGearOut.Execute := FALSE;
END_METHOD

PROPERTY PUBLIC Acceleration : mc_lreal
GET
Acceleration := mcGearIn.Acceleration;
END_GET
SET
mcGearIn.Acceleration := Acceleration;
END_SET
END_PROPERTY

PROPERTY Busy : BOOL
GET
Busy := mcGearIn.Busy OR mcGearOut.Busy;
END_GET
END_PROPERTY

METHOD Cycle : Base_Library.HRESULT
IF _AxisMaster <> 0 AND _AxisSlave <> 0 THEN
	mcGearIn(Master := _AxisMaster.AxisRef, Slave := _AxisSlave.AxisRef);
	mcGearOut(Slave := _AxisSlave.AxisRef);
END_IF
mcGearIn.Execute := FALSE;
mcGearOut.Execute := FALSE;
END_METHOD

PROPERTY PUBLIC Deceleration : mc_lreal
GET
Deceleration := mcGearIn.Deceleration;
END_GET
SET
mcGearIn.Deceleration := Deceleration;
END_SET
END_PROPERTY

PROPERTY Done : BOOL
GET
Done := not mcGearIn.Busy OR NOT mcGearOut.Busy;
END_GET
END_PROPERTY

PROPERTY Error : BOOL
GET
Error := mcGearIn.Error OR mcGearOut.Error;
END_GET
END_PROPERTY

METHOD GearIn : HRESULT
VAR_INPUT
END_VAR
IF _AxisSlave <> 0 OR _AxisMaster <> 0 THEN 
	IF _AxisSlave.IsStationary AND NOT _AxisSlave.IsCoupled AND NOT mcGearIn.Execute THEN
		mcGearIn.Execute := TRUE;
	ELSE
		GearIn := -1;
	END_IF
ELSE
	GearIn := -2;
END_IF
END_METHOD

METHOD GearOut : HRESULT
VAR_INPUT
END_VAR
IF _AxisSlave <> 0 OR _AxisMaster <> 0 THEN 
	IF _AxisSlave.IsStationary AND _AxisSlave.IsCoupled AND NOT mcGearOut.Execute THEN
		mcGearOut.Execute := TRUE;
	ELSE
		GearOut := -1;
	END_IF
END_IF
END_METHOD

PROPERTY InGear : BOOL
GET
InGear := mcGearIn.InGear AND _AxisSlave.isCoupled;
END_GET
END_PROPERTY

PROPERTY PUBLIC Jerk : mc_lreal
GET
Jerk := mcGearIn.Jerk;
END_GET
SET
mcGearIn.Jerk := Jerk;
END_SET
END_PROPERTY

PROPERTY Master : I_AxisBase
GET
Master := _AxisMaster;
END_GET
SET
_AxisMaster := Master;
END_SET
END_PROPERTY

METHOD RegisterWithParent
VAR_INPUT
	Parent	: I_HostObjects;
END_VAR
Parent.RegisterAbortable(THIS^);
Parent.RegisterCyclic(THIS^);
END_METHOD

PROPERTY Slave : I_AxisBase
GET
Slave := _AxisSlave;
END_GET
SET
_AxisSlave := Slave;
END_SET
END_PROPERTY

END_FUNCTION_BLOCK

// ---- Project Information/F_GetCompany.TcPOU
// This function has been automatically generated from the project information.
{attribute 'signature_flag' := '1073741824'}
{attribute 'TcGenerated'}
{attribute 'no-analysis'}
FUNCTION F_GetCompany : WSTRING
VAR_INPUT
	
END_VAR

F_GetCompany := "Beckhoff UK";

END_FUNCTION

// ---- Project Information/F_GetTitle.TcPOU
// This function has been automatically generated from the project information.
{attribute 'signature_flag' := '1073741824'}
{attribute 'TcGenerated'}
{attribute 'no-analysis'}
FUNCTION F_GetTitle : WSTRING
VAR_INPUT
	
END_VAR

F_GetTitle := "Motion Library";

END_FUNCTION

// ---- Project Information/F_GetVersion.TcPOU
// This function has been automatically generated from the project information.
{attribute 'signature_flag' := '1073741824'}
{attribute 'TcGenerated'}
{attribute 'no-analysis'}
FUNCTION F_GetVersion : ST_LibVersion
VAR_INPUT
	
END_VAR

F_GetVersion.iMajor := 4;
F_GetVersion.iMinor := 1;
F_GetVersion.iBuild := 1;
F_GetVersion.iRevision := 0;
F_GetVersion.sVersion := '4.1.1';
F_GetVersion.nFlags := 0;

END_FUNCTION

// ---- Tasks/SoEResetTask.TcPOU
FUNCTION_BLOCK SoEResetTask IMPLEMENTS I_Task, I_Cyclic, I_Object, I_Abortable, I_Abortable, I_Resettable
VAR
	fbSoEReset : FB_SoEReset;
	mcReset : Tc2_MC2.MC_Reset;
	_Axis : REFERENCE TO Tc2_MC2.AXIS_REF;
	State: INT;
END_VAR

METHOD Abort : HRESULT
fbSoEReset.Execute := FALSE;
mcReset.Execute := FALSE;
State := 0;
END_METHOD

PROPERTY AxisRef : reference to Axis_Ref
GET // PUBLIC
AxisRef REF= _Axis;
END_GET
SET
_Axis REF= AxisRef;
END_SET
END_PROPERTY

PROPERTY Busy : BOOL
GET
Busy := fbSoEReset.Busy;
END_GET
END_PROPERTY

METHOD Cycle : HRESULT
IF NOT __ISVALIDREF(_Axis) THEN
	Cycle := -1;
	RETURN;
END_IF

CASE State OF
	10:
		fbSoEReset.Execute := TRUE;
		State := State + 10;
	20:
		IF NOT fbSoEReset.Busy THEN
			State := State + 10;
		END_IF
	30:
		mcReset.Execute := TRUE;
		State := State + 10;
	40:
		IF mcReset.Done THEN
			State := 0;
		END_IF
END_CASE

mcReset(Axis := _Axis);
mcReset.Execute := FALSE;
fbSoEReset(Axis := _Axis);
fbSoEReset.Execute := FALSE;
END_METHOD

PROPERTY Done : BOOL
GET
Done := NOT fbSoEReset.Busy;
END_GET
END_PROPERTY

PROPERTY Error : BOOL
GET
Error := fbSoEReset.Error;
END_GET
END_PROPERTY

METHOD RegisterWithParent
VAR_INPUT
	Parent	: I_HostObjects;
END_VAR
Parent.RegisterAbortable(THIS^);
Parent.RegisterCyclic(THIS^);
Parent.RegisterTask(THIS^);
Parent.RegisterResettable(THIS^);
END_METHOD

METHOD Reset : HRESULT
IF State <> 0 THEN
	Reset := -1;
	RETURN;
END_IF
State := 10;
END_METHOD

END_FUNCTION_BLOCK
